// TIA Portal V16 export
// export: Created 2024-05-10T06:46:43.2579107Z, ExportSetting WithDefaults, DisplayName Totally Integrated Automation Portal, DisplayVersion V16, DisplayName TIA Portal Version Control Interface, DisplayVersion V16, DisplayName TIA Portal Openness, DisplayVersion V16, DisplayName STEP 7 Professional, DisplayVersion V16, DisplayName STEP 7 Safety, DisplayVersion V16, DisplayName WinCC Professional, DisplayVersion V16
DATA_BLOCK "K03_状态_DB"   // DB3
VERSION : 0.1
// stored: AutoNumber true, DBAccessibleFromOPCUA true, InstanceOfName K03_状态, InstanceOfType FB
"K03_状态"
   // VAR
   //    放行延迟 : IEC_TIMER;
   // END_VAR
BEGIN
END_DATA_BLOCK
